% RSLogix 500 project F_R_MOT_BAK002.RSS, saved by version 8.30.00.16 %
PROJECT "F_R_MOT"    % processor: Bul.1763 MicroLogix 1100 Series B %

PROGRAM FILES
  LAD 2   3 rungs

DATA FILES
  O0 OUTPUT  4 elements
  I1 INPUT  6 elements
  S2 STATUS  66 elements
  B3 BINARY  1 elements
  T4 TIMER  1 elements
  C5 COUNTER  1 elements
  R6 CONTROL  1 elements
  N7 INTEGER  1 elements
  F8 FLOAT  1 elements

LADDER 2
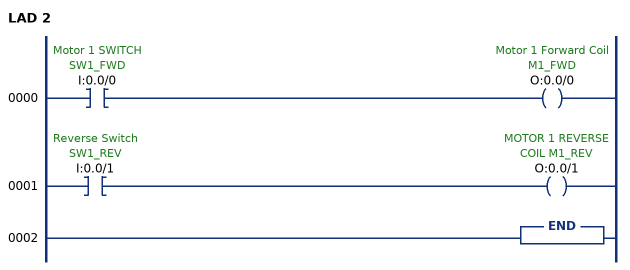
% Rung: 0 %
SOR XIC I:0.0/0 OTE O:0.0/0 EOR
%   I:0.0/0  SW1_FWD  "Motor 1 SWITCH" %
%   O:0.0/0  M1_FWD  "Motor 1 Forward Coil" %
% Rung: 1 %
SOR XIC I:0.0/1 OTE O:0.0/1 EOR
%   I:0.0/1  SW1_REV  "Reverse Switch" %
%   O:0.0/1  M1_REV  "MOTOR 1 REVERSE COIL" %
% Rung: 2 %
SOR END EOR
